Staubli VAL3: Energize.pgx

program Energize(bool cde)
  local bool cdeOn
begin
//*******************************************************************************
//*   ______
//*  / _____) /|
//* | |      / /
//* | | /\  / /
//* | | \ \/ /  _      Copyright (c) KEOLABS, 2016
//* | |  \__/  | |        http://www.keolabs.com
//* | |________| |
//*  \__________/
//*
//********************************************************************************
//*@file          : Energize
//*@author        : Yves Ragot
//*@version       : $Id: Energize.pgx 1198 2016-10-07 06:48:14Z yves $
//*@brief         : Energize the arm or not
//*
//*******************************************************************************/

  if (cde)
      // power
      enablePower()
      wait(isPowered() == true)
  else
      disablePower()
      wait(isPowered() == false)
  endIf
end
